% RSLogix 500 project QUESTAO_1_BAK180.RSS %
PROJECT "SLC00000"    % processor: type code 40 %

PROGRAM FILES
  LAD 2   7 rungs
  LAD 3 "QUESTAO_1"  6 rungs  % Contole de bomba/nivel de tanque %
  LAD 4 "QUESTAO_2"  3 rungs  % Controle de Relé-botoeira %
  LAD 5 "QUESTAO_3"  3 rungs  % Controle da prensa atraves da botoeira/timer. %
  LAD 6 "QUESTAO_4"  3 rungs  % Controle da esteira das garrafas. %
  LAD 7 "QUESTAO_5"  5 rungs  % Detecção de borda de subida e descida de sinal. %
  LAD 8 "QUESTAO_6"  6 rungs  % Máquina de solda. %
  LAD 9 "QUESTAO_7"  5 rungs  % Pisca-pisca de período de 5 segundos. %
  LAD 10 "QUESTAO_8"  4 rungs  % Sensor de presença em esteira de peças. %
  LAD 11 "QUESTAO_9"  5 rungs  % Acionamento de lâmpada aos múltiplos de cinco. %
  LAD 12 "SEMAFORO"  7 rungs  % Controle de semaforo em avenidas. %
  LAD 13 "MOTORES"  7 rungs  % Acionamento sequencial de motores. %
  LAD 14 "5_SEMTIMER"  4 rungs  % Detecção de borda de subida e descida de sinal. %

DATA FILES
  O0 SAÍDA  2 elements
  I1 ENTRADA  2 elements
  S2 STATUS  164 elements
  B3 BINÁRIO  1 elements
  T4 TEMPORIZADOR  9 elements
  C5 CONTADOR  1 elements
  R6 CONTROLE  1 elements
  N7 NÚM. INTEIRO  1 elements
  F8 PONTO FLUTUANTE  1 elements

LADDER 2
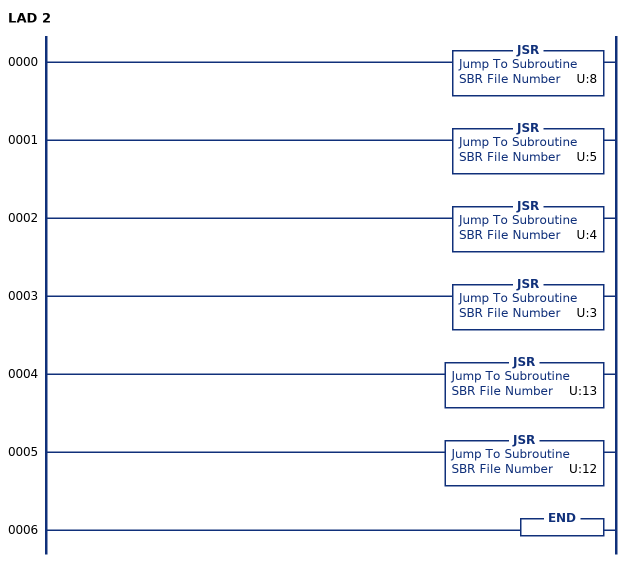
% Rung: 0 %
SOR JSR U:8 EOR
% Rung: 1 %
SOR JSR U:5 EOR
% Rung: 2 %
SOR JSR U:4 EOR
% Rung: 3 %
SOR JSR U:3 EOR
% Rung: 4 %
SOR JSR U:13 EOR
% Rung: 5 %
SOR JSR U:12 EOR
% Rung: 6 %
SOR END EOR

LADDER 3 "QUESTAO_1"    % Contole de bomba/nivel de tanque %
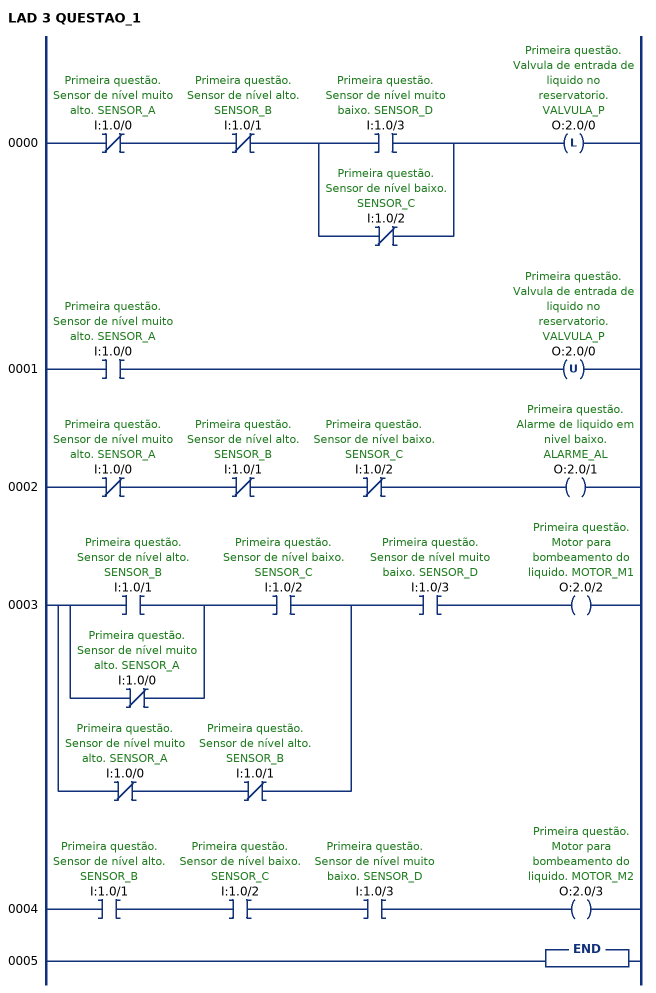
% Rung: 0 %
SOR XIO I:1.0/0 XIO I:1.0/1 BST XIC I:1.0/3 NXB XIO I:1.0/2 BND OTL O:2.0/0 EOR
%   I:1.0/0  SENSOR_A  "Primeira questão. Sensor de nível muito alto." %
%   I:1.0/1  SENSOR_B  "Primeira questão. Sensor de nível alto." %
%   I:1.0/3  SENSOR_D  "Primeira questão. Sensor de nível muito baixo." %
%   I:1.0/2  SENSOR_C  "Primeira questão. Sensor de nível baixo." %
%   O:2.0/0  VALVULA_P  "Primeira questão. Valvula de entrada de liquido no reservatorio." %
% Rung: 1 %
SOR XIC I:1.0/0 OTU O:2.0/0 EOR
%   I:1.0/0  SENSOR_A  "Primeira questão. Sensor de nível muito alto." %
%   O:2.0/0  VALVULA_P  "Primeira questão. Valvula de entrada de liquido no reservatorio." %
% Rung: 2 %
SOR XIO I:1.0/0 XIO I:1.0/1 XIO I:1.0/2 OTE O:2.0/1 EOR
%   I:1.0/0  SENSOR_A  "Primeira questão. Sensor de nível muito alto." %
%   I:1.0/1  SENSOR_B  "Primeira questão. Sensor de nível alto." %
%   I:1.0/2  SENSOR_C  "Primeira questão. Sensor de nível baixo." %
%   O:2.0/1  ALARME_AL  "Primeira questão. Alarme de liquido em nivel baixo." %
% Rung: 3 %
SOR BST BST XIC I:1.0/1 NXB XIO I:1.0/0 BND XIC I:1.0/2 NXB XIO I:1.0/0 XIO I:1.0/1 BND XIC I:1.0/3 OTE O:2.0/2 EOR
%   I:1.0/1  SENSOR_B  "Primeira questão. Sensor de nível alto." %
%   I:1.0/0  SENSOR_A  "Primeira questão. Sensor de nível muito alto." %
%   I:1.0/2  SENSOR_C  "Primeira questão. Sensor de nível baixo." %
%   I:1.0/3  SENSOR_D  "Primeira questão. Sensor de nível muito baixo." %
%   O:2.0/2  MOTOR_M1  "Primeira questão. Motor para bombeamento do liquido." %
% Rung: 4 %
SOR XIC I:1.0/1 XIC I:1.0/2 XIC I:1.0/3 OTE O:2.0/3 EOR
%   I:1.0/1  SENSOR_B  "Primeira questão. Sensor de nível alto." %
%   I:1.0/2  SENSOR_C  "Primeira questão. Sensor de nível baixo." %
%   I:1.0/3  SENSOR_D  "Primeira questão. Sensor de nível muito baixo." %
%   O:2.0/3  MOTOR_M2  "Primeira questão. Motor para bombeamento do liquido." %
% Rung: 5 %
SOR END EOR

LADDER 4 "QUESTAO_2"    % Controle de Relé-botoeira %
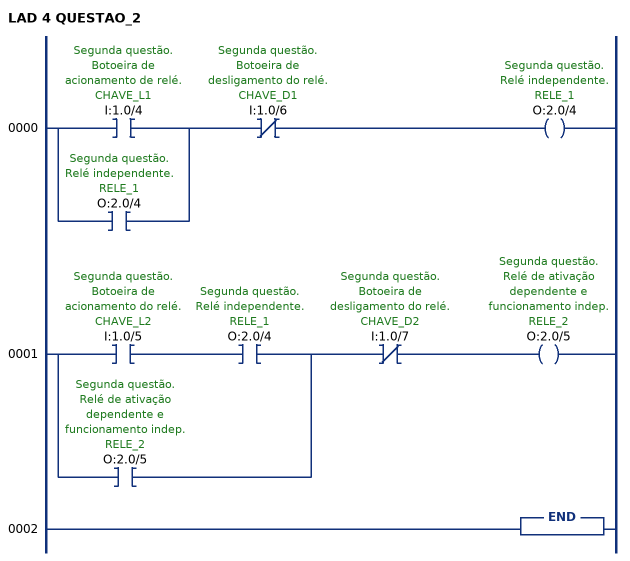
% Rung: 0 %
SOR BST XIC I:1.0/4 NXB XIC O:2.0/4 BND XIO I:1.0/6 OTE O:2.0/4 EOR
%   I:1.0/4  CHAVE_L1  "Segunda questão. Botoeira de acionamento de relé." %
%   O:2.0/4  RELE_1  "Segunda questão. Relé independente." %
%   I:1.0/6  CHAVE_D1  "Segunda questão. Botoeira de desligamento do relé." %
% Rung: 1 %
SOR BST XIC I:1.0/5 XIC O:2.0/4 NXB XIC O:2.0/5 BND XIO I:1.0/7 OTE O:2.0/5 EOR
%   I:1.0/5  CHAVE_L2  "Segunda questão. Botoeira de acionamento do relé." %
%   O:2.0/4  RELE_1  "Segunda questão. Relé independente." %
%   O:2.0/5  RELE_2  "Segunda questão. Relé de ativação dependente e funcionamento indep." %
%   I:1.0/7  CHAVE_D2  "Segunda questão. Botoeira de desligamento do relé." %
% Rung: 2 %
SOR END EOR

LADDER 5 "QUESTAO_3"    % Controle da prensa atraves da botoeira/timer. %
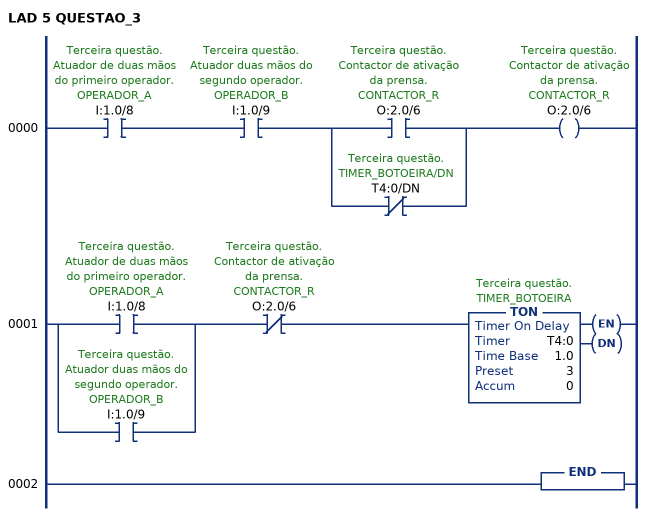
% Rung: 0 %
SOR XIC I:1.0/8 XIC I:1.0/9 BST XIC O:2.0/6 NXB XIO T4:0/DN BND OTE O:2.0/6 EOR
%   I:1.0/8  OPERADOR_A  "Terceira questão. Atuador de duas mãos do primeiro operador." %
%   I:1.0/9  OPERADOR_B  "Terceira questão. Atuador duas mãos do segundo operador." %
%   O:2.0/6  CONTACTOR_R  "Terceira questão. Contactor de ativação da prensa." %
%   T4:0  TIMER_BOTOEIRA  "Terceira questão." %
% Rung: 1 %
SOR BST XIC I:1.0/8 NXB XIC I:1.0/9 BND XIO O:2.0/6 TON T4:0 1.0 3 0 EOR
%   I:1.0/8  OPERADOR_A  "Terceira questão. Atuador de duas mãos do primeiro operador." %
%   I:1.0/9  OPERADOR_B  "Terceira questão. Atuador duas mãos do segundo operador." %
%   O:2.0/6  CONTACTOR_R  "Terceira questão. Contactor de ativação da prensa." %
%   T4:0  TIMER_BOTOEIRA  "Terceira questão." %
% Rung: 2 %
SOR END EOR

LADDER 6 "QUESTAO_4"    % Controle da esteira das garrafas. %
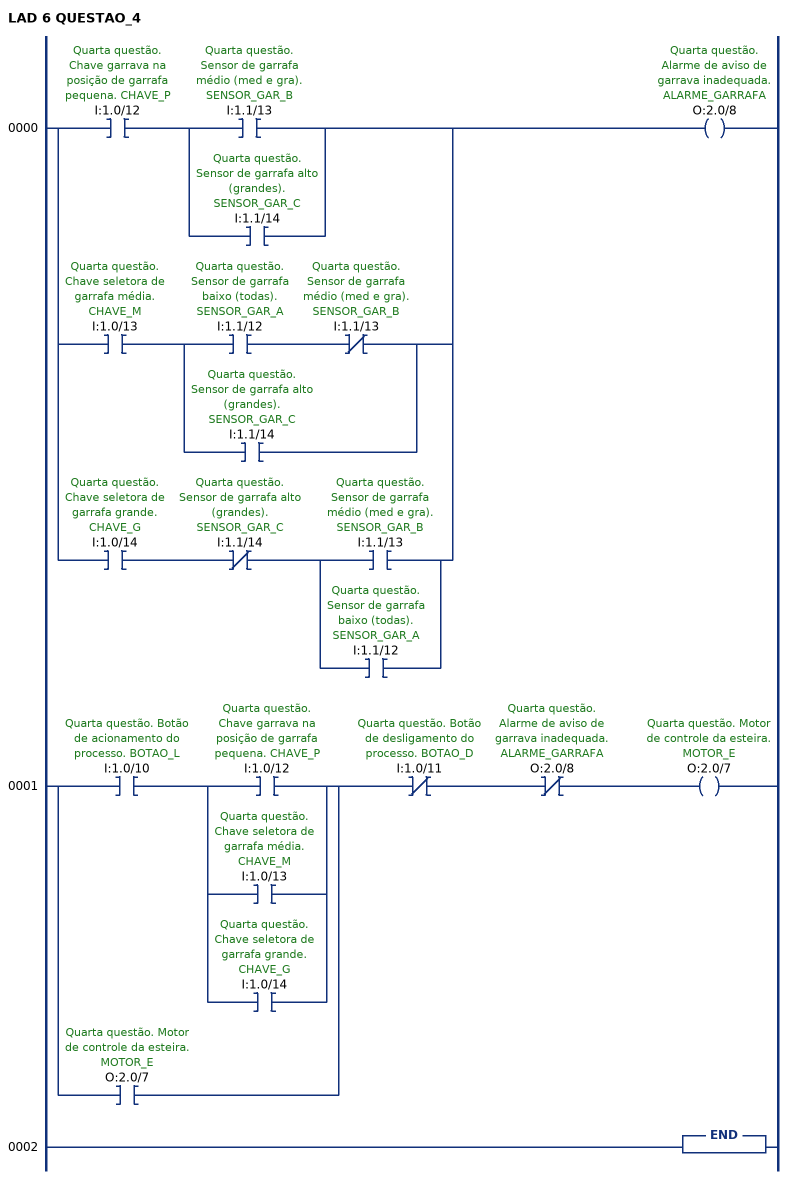
% Rung: 0 %
SOR BST XIC I:1.0/12 BST XIC I:1.1/13 NXB XIC I:1.1/14 BND NXB BST XIC I:1.0/13 BST XIC I:1.1/12 XIO I:1.1/13 NXB XIC I:1.1/14 BND NXB XIC I:1.0/14 XIO I:1.1/14 BST XIC I:1.1/13 NXB XIC I:1.1/12 BND BND BND OTE O:2.0/8 EOR
%   I:1.0/12  CHAVE_P  "Quarta questão. Chave garrava na posição de garrafa pequena." %
%   I:1.1/13  SENSOR_GAR_B  "Quarta questão. Sensor de garrafa médio (med e gra)." %
%   I:1.1/14  SENSOR_GAR_C  "Quarta questão. Sensor de garrafa alto (grandes)." %
%   I:1.0/13  CHAVE_M  "Quarta questão. Chave seletora de garrafa média." %
%   I:1.1/12  SENSOR_GAR_A  "Quarta questão. Sensor de garrafa baixo (todas)." %
%   I:1.0/14  CHAVE_G  "Quarta questão. Chave seletora de garrafa grande." %
%   O:2.0/8  ALARME_GARRAFA  "Quarta questão. Alarme de aviso de garrava inadequada." %
% Rung: 1 %
SOR BST XIC I:1.0/10 BST XIC I:1.0/12 NXB BST XIC I:1.0/13 NXB XIC I:1.0/14 BND BND NXB XIC O:2.0/7 BND XIO I:1.0/11 XIO O:2.0/8 OTE O:2.0/7 EOR
%   I:1.0/10  BOTAO_L  "Quarta questão. Botão de acionamento do processo." %
%   I:1.0/12  CHAVE_P  "Quarta questão. Chave garrava na posição de garrafa pequena." %
%   I:1.0/13  CHAVE_M  "Quarta questão. Chave seletora de garrafa média." %
%   I:1.0/14  CHAVE_G  "Quarta questão. Chave seletora de garrafa grande." %
%   O:2.0/7  MOTOR_E  "Quarta questão. Motor de controle da esteira." %
%   I:1.0/11  BOTAO_D  "Quarta questão. Botão de desligamento do processo." %
%   O:2.0/8  ALARME_GARRAFA  "Quarta questão. Alarme de aviso de garrava inadequada." %
% Rung: 2 %
SOR END EOR

LADDER 7 "QUESTAO_5"    % Detecção de borda de subida e descida de sinal. %
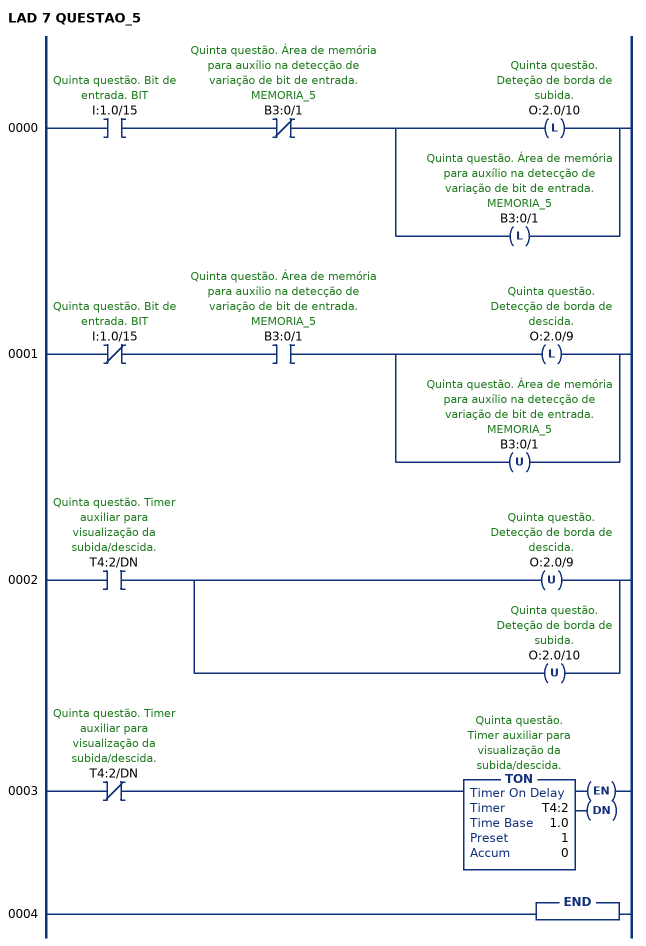
% Rung: 0 %
SOR XIC I:1.0/15 XIO B3:0/1 BST OTL O:2.0/10 NXB OTL B3:0/1 BND EOR
%   I:1.0/15  BIT  "Quinta questão. Bit de entrada." %
%   B3:0/1  MEMORIA_5  "Quinta questão. Área de memória para auxílio na detecção de variação de bit de entrada." %
%   O:2.0/10  "Quinta questão. Deteção de borda de subida." %
% Rung: 1 %
SOR XIO I:1.0/15 XIC B3:0/1 BST OTL O:2.0/9 NXB OTU B3:0/1 BND EOR
%   I:1.0/15  BIT  "Quinta questão. Bit de entrada." %
%   B3:0/1  MEMORIA_5  "Quinta questão. Área de memória para auxílio na detecção de variação de bit de entrada." %
%   O:2.0/9  "Quinta questão. Detecção de borda de descida." %
% Rung: 2 %
SOR XIC T4:2/DN BST OTU O:2.0/9 NXB OTU O:2.0/10 BND EOR
%   T4:2  "Quinta questão. Timer auxiliar para visualização da subida/descida." %
%   O:2.0/9  "Quinta questão. Detecção de borda de descida." %
%   O:2.0/10  "Quinta questão. Deteção de borda de subida." %
% Rung: 3 %
SOR XIO T4:2/DN TON T4:2 1.0 1 0 EOR
%   T4:2  "Quinta questão. Timer auxiliar para visualização da subida/descida." %
% Rung: 4 %
SOR END EOR

LADDER 8 "QUESTAO_6"    % Máquina de solda. %
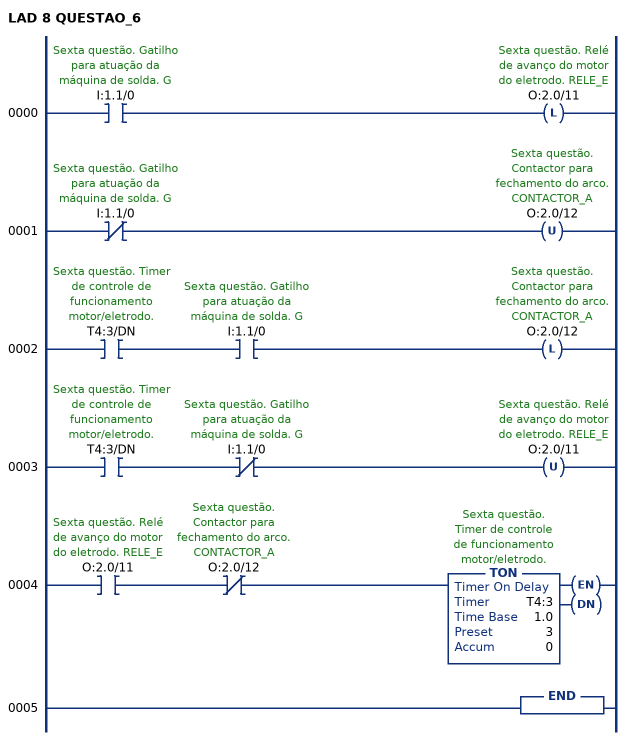
% Rung: 0 %
SOR XIC I:1.1/0 OTL O:2.0/11 EOR
%   I:1.1/0  G  "Sexta questão. Gatilho para atuação da máquina de solda." %
%   O:2.0/11  RELE_E  "Sexta questão. Relé de avanço do motor do eletrodo." %
% Rung: 1 %
SOR XIO I:1.1/0 OTU O:2.0/12 EOR
%   I:1.1/0  G  "Sexta questão. Gatilho para atuação da máquina de solda." %
%   O:2.0/12  CONTACTOR_A  "Sexta questão. Contactor para fechamento do arco." %
% Rung: 2 %
SOR XIC T4:3/DN XIC I:1.1/0 OTL O:2.0/12 EOR
%   T4:3  "Sexta questão. Timer de controle de funcionamento motor/eletrodo." %
%   I:1.1/0  G  "Sexta questão. Gatilho para atuação da máquina de solda." %
%   O:2.0/12  CONTACTOR_A  "Sexta questão. Contactor para fechamento do arco." %
% Rung: 3 %
SOR XIC T4:3/DN XIO I:1.1/0 OTU O:2.0/11 EOR
%   T4:3  "Sexta questão. Timer de controle de funcionamento motor/eletrodo." %
%   I:1.1/0  G  "Sexta questão. Gatilho para atuação da máquina de solda." %
%   O:2.0/11  RELE_E  "Sexta questão. Relé de avanço do motor do eletrodo." %
% Rung: 4 %
SOR XIC O:2.0/11 XIO O:2.0/12 TON T4:3 1.0 3 0 EOR
%   O:2.0/11  RELE_E  "Sexta questão. Relé de avanço do motor do eletrodo." %
%   O:2.0/12  CONTACTOR_A  "Sexta questão. Contactor para fechamento do arco." %
%   T4:3  "Sexta questão. Timer de controle de funcionamento motor/eletrodo." %
% Rung: 5 %
SOR END EOR

LADDER 9 "QUESTAO_7"    % Pisca-pisca de período de 5 segundos. %
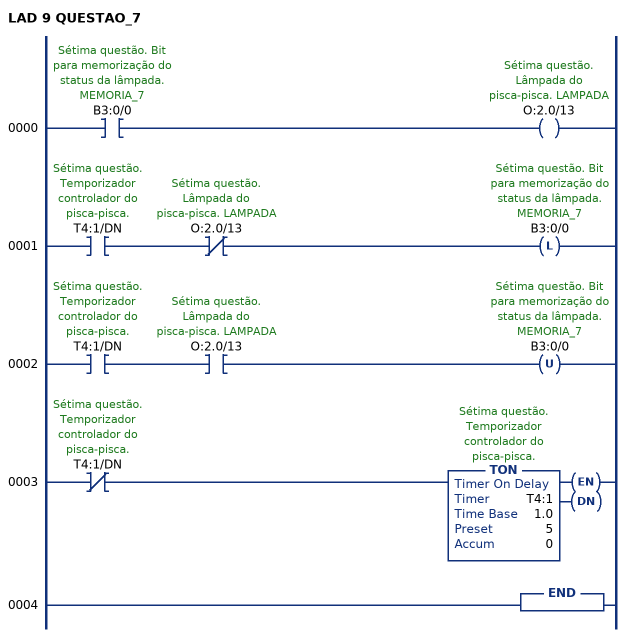
% Rung: 0 %
SOR XIC B3:0/0 OTE O:2.0/13 EOR
%   B3:0/0  MEMORIA_7  "Sétima questão. Bit para memorização do status da lâmpada." %
%   O:2.0/13  LAMPADA  "Sétima questão. Lâmpada do pisca-pisca." %
% Rung: 1 %
SOR XIC T4:1/DN XIO O:2.0/13 OTL B3:0/0 EOR
%   T4:1  "Sétima questão. Temporizador controlador do pisca-pisca." %
%   O:2.0/13  LAMPADA  "Sétima questão. Lâmpada do pisca-pisca." %
%   B3:0/0  MEMORIA_7  "Sétima questão. Bit para memorização do status da lâmpada." %
% Rung: 2 %
SOR XIC T4:1/DN XIC O:2.0/13 OTU B3:0/0 EOR
%   T4:1  "Sétima questão. Temporizador controlador do pisca-pisca." %
%   O:2.0/13  LAMPADA  "Sétima questão. Lâmpada do pisca-pisca." %
%   B3:0/0  MEMORIA_7  "Sétima questão. Bit para memorização do status da lâmpada." %
% Rung: 3 %
SOR XIO T4:1/DN TON T4:1 1.0 5 0 EOR
%   T4:1  "Sétima questão. Temporizador controlador do pisca-pisca." %
% Rung: 4 %
SOR END EOR

LADDER 10 "QUESTAO_8"    % Sensor de presença em esteira de peças. %
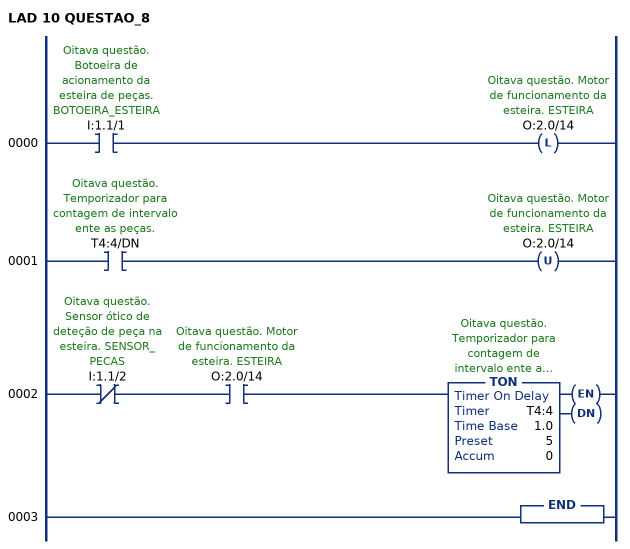
% Rung: 0 %
SOR XIC I:1.1/1 OTL O:2.0/14 EOR
%   I:1.1/1  BOTOEIRA_ESTEIRA  "Oitava questão. Botoeira de acionamento da esteira de peças." %
%   O:2.0/14  ESTEIRA  "Oitava questão. Motor de funcionamento da esteira." %
% Rung: 1 %
SOR XIC T4:4/DN OTU O:2.0/14 EOR
%   T4:4  "Oitava questão. Temporizador para contagem de intervalo ente as peças." %
%   O:2.0/14  ESTEIRA  "Oitava questão. Motor de funcionamento da esteira." %
% Rung: 2 %
SOR XIO I:1.1/2 XIC O:2.0/14 TON T4:4 1.0 5 0 EOR
%   I:1.1/2  SENSOR_PECAS  "Oitava questão. Sensor ótico de deteção de peça na esteira." %
%   O:2.0/14  ESTEIRA  "Oitava questão. Motor de funcionamento da esteira." %
%   T4:4  "Oitava questão. Temporizador para contagem de intervalo ente as peças." %
% Rung: 3 %
SOR END EOR

LADDER 11 "QUESTAO_9"    % Acionamento de lâmpada aos múltiplos de cinco. %
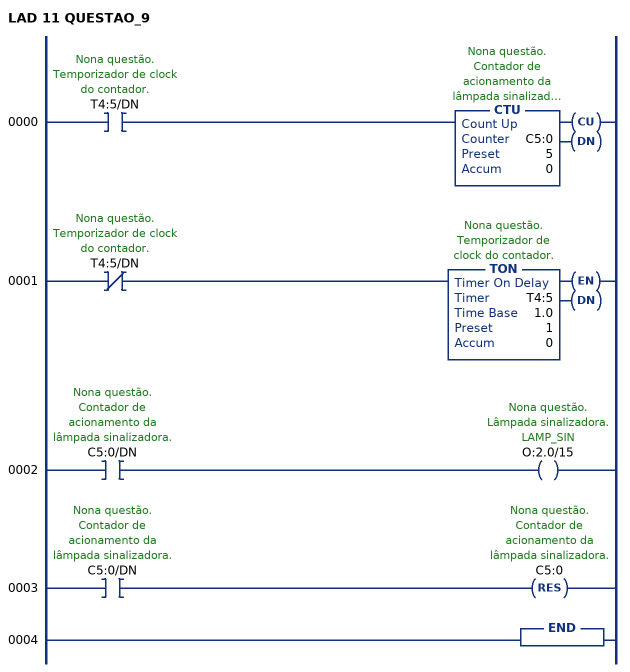
% Rung: 0 %
SOR XIC T4:5/DN CTU C5:0 5 0 EOR
%   T4:5  "Nona questão. Temporizador de clock do contador." %
%   C5:0  "Nona questão. Contador de acionamento da lâmpada sinalizadora." %
% Rung: 1 %
SOR XIO T4:5/DN TON T4:5 1.0 1 0 EOR
%   T4:5  "Nona questão. Temporizador de clock do contador." %
% Rung: 2 %
SOR XIC C5:0/DN OTE O:2.0/15 EOR
%   C5:0  "Nona questão. Contador de acionamento da lâmpada sinalizadora." %
%   O:2.0/15  LAMP_SIN  "Nona questão. Lâmpada sinalizadora." %
% Rung: 3 %
SOR XIC C5:0/DN RES C5:0 EOR
%   C5:0  "Nona questão. Contador de acionamento da lâmpada sinalizadora." %
% Rung: 4 %
SOR END EOR

LADDER 12 "SEMAFORO"    % Controle de semaforo em avenidas. %
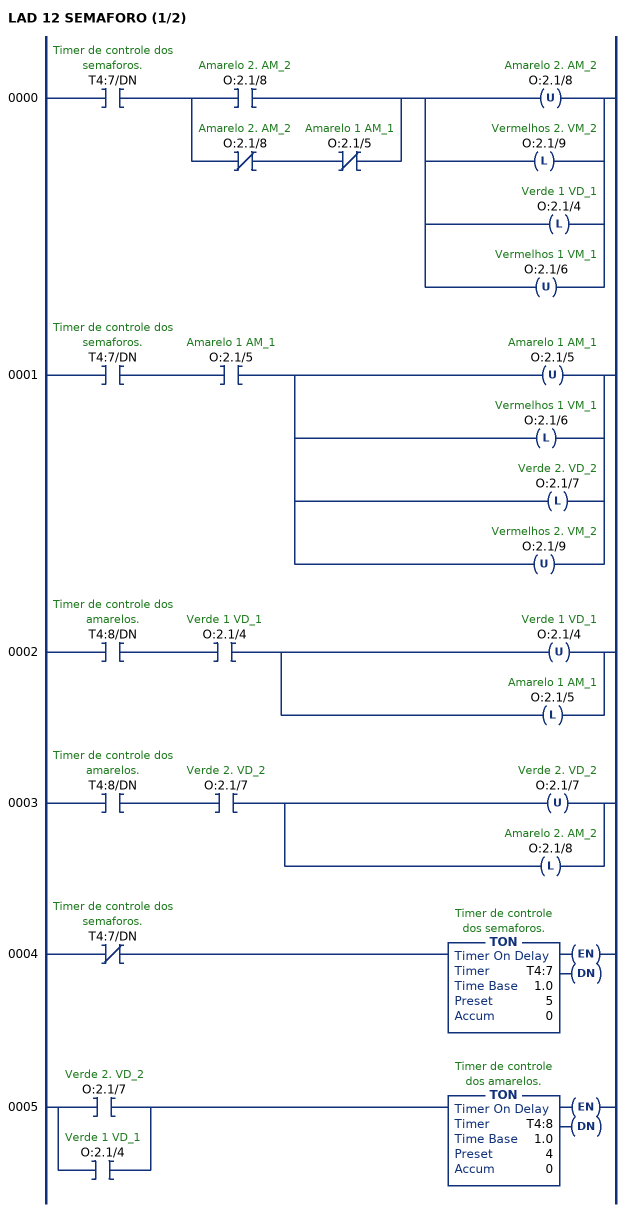
% Rung: 0 %
SOR XIC T4:7/DN BST XIC O:2.1/8 NXB XIO O:2.1/8 XIO O:2.1/5 BND BST OTU O:2.1/8 NXB BST OTL O:2.1/9 NXB BST OTL O:2.1/4 NXB OTU O:2.1/6 BND BND BND EOR
%   T4:7  "Timer de controle dos semaforos." %
%   O:2.1/8  AM_2  "Amarelo 2." %
%   O:2.1/5  AM_1  "Amarelo 1" %
%   O:2.1/9  VM_2  "Vermelhos 2." %
%   O:2.1/4  VD_1  "Verde 1" %
%   O:2.1/6  VM_1  "Vermelhos 1" %
% Rung: 1 %
SOR XIC T4:7/DN XIC O:2.1/5 BST OTU O:2.1/5 NXB BST OTL O:2.1/6 NXB BST OTL O:2.1/7 NXB OTU O:2.1/9 BND BND BND EOR
%   T4:7  "Timer de controle dos semaforos." %
%   O:2.1/5  AM_1  "Amarelo 1" %
%   O:2.1/6  VM_1  "Vermelhos 1" %
%   O:2.1/7  VD_2  "Verde 2." %
%   O:2.1/9  VM_2  "Vermelhos 2." %
% Rung: 2 %
SOR XIC T4:8/DN XIC O:2.1/4 BST OTU O:2.1/4 NXB OTL O:2.1/5 BND EOR
%   T4:8  "Timer de controle dos amarelos." %
%   O:2.1/4  VD_1  "Verde 1" %
%   O:2.1/5  AM_1  "Amarelo 1" %
% Rung: 3 %
SOR XIC T4:8/DN XIC O:2.1/7 BST OTU O:2.1/7 NXB OTL O:2.1/8 BND EOR
%   T4:8  "Timer de controle dos amarelos." %
%   O:2.1/7  VD_2  "Verde 2." %
%   O:2.1/8  AM_2  "Amarelo 2." %
% Rung: 4 %
SOR XIO T4:7/DN TON T4:7 1.0 5 0 EOR
%   T4:7  "Timer de controle dos semaforos." %
% Rung: 5 %
SOR BST XIC O:2.1/7 NXB XIC O:2.1/4 BND TON T4:8 1.0 4 0 EOR
%   O:2.1/7  VD_2  "Verde 2." %
%   O:2.1/4  VD_1  "Verde 1" %
%   T4:8  "Timer de controle dos amarelos." %

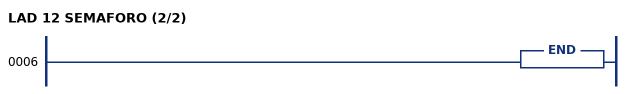
% Rung: 6 %
SOR END EOR

LADDER 13 "MOTORES"    % Acionamento sequencial de motores. %
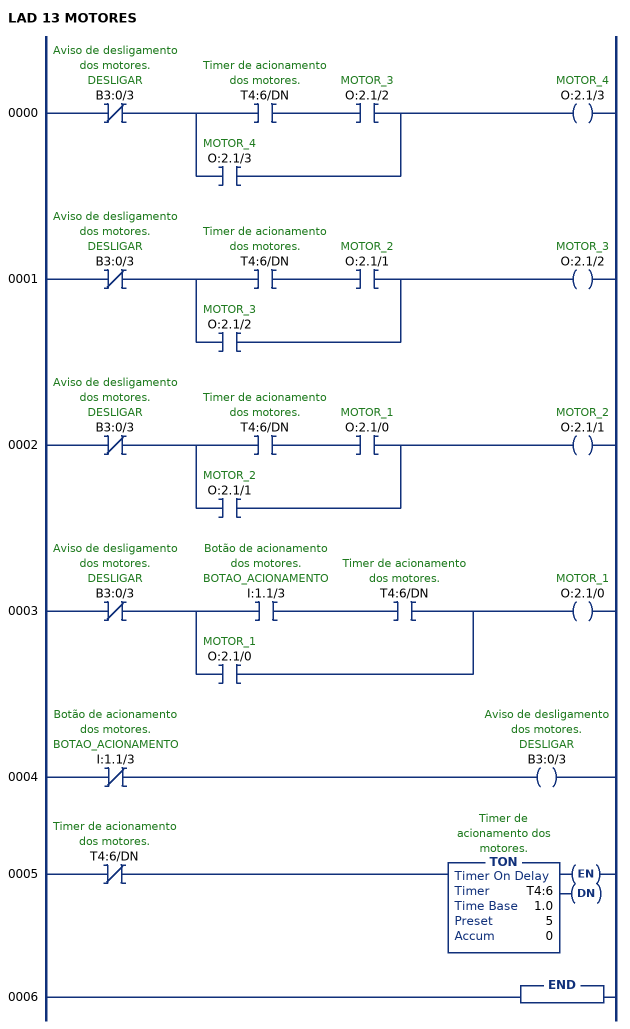
% Rung: 0 %
SOR XIO B3:0/3 BST XIC T4:6/DN XIC O:2.1/2 NXB XIC O:2.1/3 BND OTE O:2.1/3 EOR
%   B3:0/3  DESLIGAR  "Aviso de desligamento dos motores." %
%   T4:6  "Timer de acionamento dos motores." %
%   O:2.1/2  MOTOR_3 %
%   O:2.1/3  MOTOR_4 %
% Rung: 1 %
SOR XIO B3:0/3 BST XIC T4:6/DN XIC O:2.1/1 NXB XIC O:2.1/2 BND OTE O:2.1/2 EOR
%   B3:0/3  DESLIGAR  "Aviso de desligamento dos motores." %
%   T4:6  "Timer de acionamento dos motores." %
%   O:2.1/1  MOTOR_2 %
%   O:2.1/2  MOTOR_3 %
% Rung: 2 %
SOR XIO B3:0/3 BST XIC T4:6/DN XIC O:2.1/0 NXB XIC O:2.1/1 BND OTE O:2.1/1 EOR
%   B3:0/3  DESLIGAR  "Aviso de desligamento dos motores." %
%   T4:6  "Timer de acionamento dos motores." %
%   O:2.1/0  MOTOR_1 %
%   O:2.1/1  MOTOR_2 %
% Rung: 3 %
SOR XIO B3:0/3 BST XIC I:1.1/3 XIC T4:6/DN NXB XIC O:2.1/0 BND OTE O:2.1/0 EOR
%   B3:0/3  DESLIGAR  "Aviso de desligamento dos motores." %
%   I:1.1/3  BOTAO_ACIONAMENTO  "Botão de acionamento dos motores." %
%   T4:6  "Timer de acionamento dos motores." %
%   O:2.1/0  MOTOR_1 %
% Rung: 4 %
SOR XIO I:1.1/3 OTE B3:0/3 EOR
%   I:1.1/3  BOTAO_ACIONAMENTO  "Botão de acionamento dos motores." %
%   B3:0/3  DESLIGAR  "Aviso de desligamento dos motores." %
% Rung: 5 %
SOR XIO T4:6/DN TON T4:6 1.0 5 0 EOR
%   T4:6  "Timer de acionamento dos motores." %
% Rung: 6 %
SOR END EOR

LADDER 14 "5_SEMTIMER"    % Detecção de borda de subida e descida de sinal. %
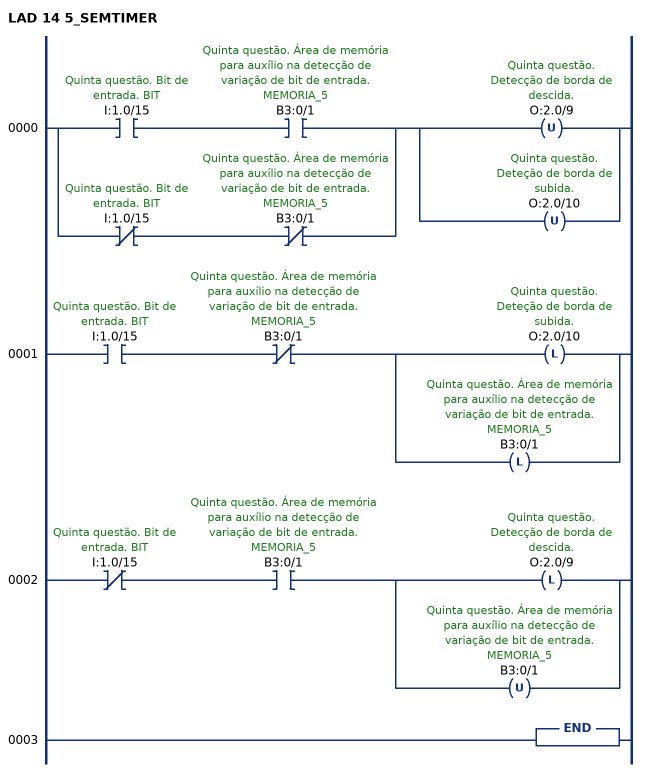
% Rung: 0 %
SOR BST XIC I:1.0/15 XIC B3:0/1 NXB XIO I:1.0/15 XIO B3:0/1 BND BST OTU O:2.0/9 NXB OTU O:2.0/10 BND EOR
%   I:1.0/15  BIT  "Quinta questão. Bit de entrada." %
%   B3:0/1  MEMORIA_5  "Quinta questão. Área de memória para auxílio na detecção de variação de bit de entrada." %
%   O:2.0/9  "Quinta questão. Detecção de borda de descida." %
%   O:2.0/10  "Quinta questão. Deteção de borda de subida." %
% Rung: 1 %
SOR XIC I:1.0/15 XIO B3:0/1 BST OTL O:2.0/10 NXB OTL B3:0/1 BND EOR
%   I:1.0/15  BIT  "Quinta questão. Bit de entrada." %
%   B3:0/1  MEMORIA_5  "Quinta questão. Área de memória para auxílio na detecção de variação de bit de entrada." %
%   O:2.0/10  "Quinta questão. Deteção de borda de subida." %
% Rung: 2 %
SOR XIO I:1.0/15 XIC B3:0/1 BST OTL O:2.0/9 NXB OTU B3:0/1 BND EOR
%   I:1.0/15  BIT  "Quinta questão. Bit de entrada." %
%   B3:0/1  MEMORIA_5  "Quinta questão. Área de memória para auxílio na detecção de variação de bit de entrada." %
%   O:2.0/9  "Quinta questão. Detecção de borda de descida." %
% Rung: 3 %
SOR END EOR

OTHER DOCUMENTED ADDRESSES
  B3:0/2  VARIACAO  "Quinta questão. Detecção de variação de bit."
  DFILE:0  "SAÍDA"
  DFILE:1  "ENTRADA"
  DFILE:2  "STATUS"
  DFILE:3  "BINÁRIO"
  DFILE:4  "TEMPORIZADOR"
  DFILE:5  "CONTADOR"
  DFILE:6  "CONTROLE"
  DFILE:7  "NÚM. INTEIRO"
  DFILE:8  "PONTO FLUTUANTE"
  Q0:0  QUESTAO_1
  Q2:0  LAD3
  T4  

REVISION NOTES
  0: Resolução da primeira questão. Implementação alfa.
  1: Implementação da segunda questão
  2: Implementação da terceira questão

DATA TABLE (non-zero values as saved)
DATA B3
% B3:0 % 0X0008
DATA T4
% .PRE .ACC %
% T4:0 % 3 0
% T4:1 % 5 0
% T4:2 % 1 0
% T4:3 % 3 0
% T4:4 % 5 0
% T4:5 % 1 0
% T4:6 % 5 0
% T4:7 % 5 0
% T4:8 % 4 0
DATA C5
% .PRE .ACC %
% C5:0 % 5 0
